// TIA Portal V19 export
VAR_GLOBAL   // PLC tag table "Equipment_Template_6"
END_VAR
